(* PLC project Unnamed, Unknown Unnamed 1 *)
(* stored: creationDateTime 2026-05-07T14:01:30, modificationDateTime 2026-05-07T14:01:30 *)

PROGRAM main
  VAR
    BtnGreen AT %IX0.0 : BOOL;
  END_VAR
  VAR
    LEDGreen : BOOL;
  END_VAR

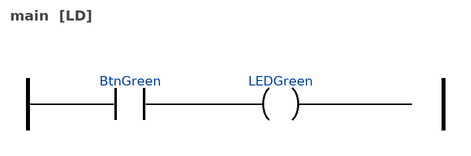
(* LD diagram, written out as Structured Text *)
LEDGreen := BtnGreen;
END_PROGRAM

CONFIGURATION Config0
  RESOURCE Res0 ON PLC
    TASK task0(INTERVAL := T#20ms, PRIORITY := 1);
    PROGRAM instance0 WITH task0 : main;
  END_RESOURCE
END_CONFIGURATION
